// TIA Portal V20 export
FUNCTION_BLOCK "CC_Vibrator_Control"   // FB103, LAD
{ S7_Optimized_Access := 'TRUE' }
// stored: AutoNumber false, MemoryReserve 100, SetENOAutomatically false
   VAR_INPUT
      StartVibrating : Bool;
      Reset : Bool;
      Axis : TO_SpeedAxis;
      tmpVelocity : LReal := 2840.0;
   END_VAR
   VAR
      MC_Power_data { S7_SetPoint := 'True'} : MC_POWER;
      MC_Reset_data { S7_SetPoint := 'True'} : MC_RESET;
      MC_MoveJog_data { S7_SetPoint := 'True'} : MC_MOVEJOG;
      MC_HALT_data { S7_SetPoint := 'True'} : MC_HALT;
   END_VAR
BEGIN

REGION Network 1: Hydraulic Unit Motion Control
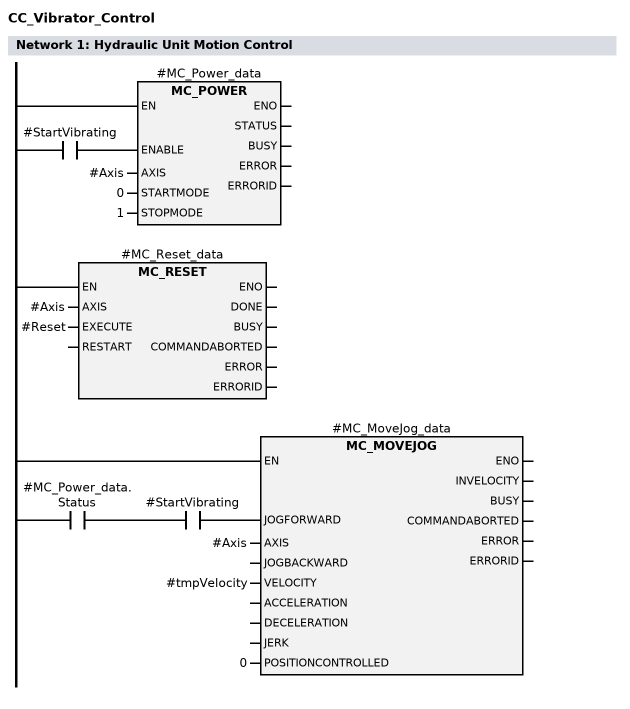
   RUNG wire#powerrail
      #MC_Power_data.MC_POWER(Enable := wire#w1, Axis := #Axis, StartMode := 0, StopMode := 1, Status =>, Busy =>, Error =>, ErrorId =>)
   END_RUNG
   RUNG wire#powerrail
      Contact( #StartVibrating )
   END_RUNG wire#w1
   RUNG wire#powerrail
      #MC_Reset_data.MC_RESET(Axis := #Axis, Execute := #Reset, Restart :=, Done =>, Busy =>, CommandAborted =>, Error =>, ErrorId =>)
   END_RUNG
   RUNG wire#powerrail
      #MC_MoveJog_data.MC_MOVEJOG(JogForward := wire#w2, Axis := #Axis, JogBackward :=, Velocity := #tmpVelocity, Acceleration :=, Deceleration :=, Jerk :=, PositionControlled := 0, InVelocity =>, Busy =>, CommandAborted =>, Error =>, ErrorId =>)
   END_RUNG
   RUNG wire#powerrail
      Contact( #MC_Power_data.Status )
      Contact( #StartVibrating )
   END_RUNG wire#w2
   // the same network as SCL:
   #MC_Power_data(Enable := #StartVibrating, Axis := #Axis, StartMode := 0, StopMode := 1);   // MC_POWER
   #MC_Reset_data(Axis := #Axis, Execute := #Reset);   // MC_RESET
   #MC_MoveJog_data(JogForward := #MC_Power_data.Status AND #StartVibrating,   // MC_MOVEJOG
                    Axis := #Axis,
                    Velocity := #tmpVelocity,
                    PositionControlled := 0);
END_REGION
END_FUNCTION_BLOCK
